// TIA Portal V19 export
ORGANIZATION_BLOCK "OBNL_FLT"   // OB85, STL, AccessError
TITLE = "Organization Block (OB) Not Loaded Fault"
   VAR_TEMP
      OB85_EV_CLASS : Byte;   // 16#35 Event class 3
      OB85_FLT_ID : Byte;   // 16#XX, Fault identification code
      OB85_PRIORITY : Byte;   // Priority of OB Execution
      OB85_OB_NUMBR : Byte;   // 85 (Organization block 85, OB85)
      OB85_RESERVED_1 : Byte;   // Reserved for system
      OB85_RESERVED_2 : Byte;   // Reserved for system
      OB85_RESERVED_3 : Int;   // Reserved for system
      OB85_ERR_EV_CLASS : Byte;   // Class of event causing error
      OB85_ERR_EV_NUM : Byte;   // Number of event causing error
      OB85_OB_PRIOR : Byte;   // Priority of OB causing error
      OB85_OB_NUM : Byte;   // Number of OB causing error
      OB85_DATE_TIME : Date_And_Time;   // Date and time OB85 started
   END_VAR
BEGIN

NETWORK
TITLE = 
      L     b#16#A1;  //
      L     #OB85_FLT_ID;
      ==I;
      JC    K_OB;
      L     b#16#A2;  //
      ==I;
      JC    K_OB;
      L     b#16#A3;  //
      L     #OB85_FLT_ID;
      ==I;
      JC    K_B;
      JU    F_PA;


NETWORK
TITLE = 
K_OB: JU    STOP;
      JU    ENDE;


NETWORK
TITLE = 
K_B:  JU    STOP;
      JU    ENDE;


NETWORK
TITLE = 
F_PA: NOP   0;
      JU    ENDE;


NETWORK
TITLE = 
STOP: CALL  STP;


NETWORK
TITLE = 

//

ENDE: NOP   0;

END_ORGANIZATION_BLOCK
